TYPE XyTableComSubscribeSegments :
STRUCT
  Start : DINT;
  End : DINT;
  Data : ARRAY[0..10] OF Segment;
END_STRUCT
END_TYPE

(* stored: Version 1.1.0.1
   DUT XyTableComSubscribeSegments: Id {4dacbee3-1536-42ac-9130-f733008dbf57} *)
